FUNCTION TryConvert_LWORD_TO_BYTE : BOOL
VAR_INPUT
	in : LWORD;
	out : REFERENCE TO BYTE;
END_VAR

IF in > DatatypeLimits.MAX_VALUE_OF_LWORD_WHICH_CAN_BE_HELD_IN_A_BYTE THEN
	RETURN;
END_IF

out := LWORD_TO_BYTE(in);
TryConvert_LWORD_TO_BYTE := TRUE;

END_FUNCTION

(* stored: Version 1.1.0.1, ProductVersion 3.1.4024.12
   POU TryConvert_LWORD_TO_BYTE: Id {c7fefa72-8fd3-4200-a54c-6107e58299e6}, SpecialFunc None *)
